	EmptyEvents				: ST_Event; // to Clear the event array[n]
	CmdEmpty				: ST_Command;
	iEventNameFailed 		: E_EventName;
	iEventName				: E_EventName;

	//nCommandNumber:UINT;
	//fbModuleIDNameCheck: FB_ModuleIDNameCheck;
	//fbParameterCheck: FB_ParameterCheck;	
END_VAR

VAR_IN_OUT
	arrRCMD 				: ARRAY [1..NO_OF_CMD_BUFFER] OF ST_Command;
	arrEvent				: ARRAY [1..NO_OF_EVENT_BUFFER] OF ST_Event;
END_VAR
//nCommandNumber := INT_TO_UINT(n);
bErr    														:= FALSE;
sStatus 														:= '';

arrEvent[n] 													:= EmptyEvents;

IF arrRCMD[n].eTaskName = E_TaskName.AlarmReset THEN
	M_nModuleIDConversion(eModuleID:=arrRCMD[n].eModuleID,iLevel=>iLevel);
	//iLevel := arrRCMD[n].iParam[1];
	//iLevel := arrRCMD[n].iParam[1]/1000;
ELSE
	M_nModuleIDConversion(eModuleID:=arrRCMD[n].eModuleID,iLevel=>iLevel);
	(*
	CASE arrRCMD[n].eModuleID OF
		E_ModuleID.TESTER_L_A_01 : iLevel:=1;
		E_ModuleID.TESTER_L_A_02 : iLevel:=2;
		E_ModuleID.TESTER_L_A_03 : iLevel:=3;
		
	END_CASE
	*)	
END_IF

IF bInvalidCommand = TRUE THEN
	bErr := TRUE; 
	sStatus := 'Invalid command received';
ELSIF iLevel = 0 THEN
	bErr := TRUE; 
	sStatus := 'Wrong Module ID';
ELSIF  arrTCShuttlePOC[iLevel].stGblParam.bAlarmOccur =TRUE THEN
	IF arrRCMD[n].eTaskName = E_TaskName.TIUSlideOut THEN 
		bErr := TRUE; 
		sStatus := 'Please clear alarm 1st';
	//ELSIF UDINT_TO_INT(arrTCVIO[iLevel].iAlarmCode) <> arrRCMD[n].iParam[1] THEN
	//	bErr := TRUE; 
	//	sStatus := concat('Alarm Code not match with current AlarmCode ', UDINT_TO_STRING(arrTCVIO[iLevel].iAlarmCode));
	END_IF
ELSIF arrRCMD[n].eTaskName = E_TaskName.TCCSessionRequest OR
   		arrRCMD[n].eTaskName = E_TaskName.DPSPower OR
   		arrRCMD[n].eTaskName = E_TaskName.TIUSlideOut THEN
			//bErr:=SEL(arrTCLevelState[iLevel] = E_State.eDisabled,FALSE,TRUE);
			//sStatus := SEL(bErr,'','Module is Disabled');
			bErr:=SEL(TC_ModuleState[iLevel].Tester = E_State.eDisabled OR 
					  TC_ModuleState[iLevel].TCSite[1].TCU = E_State.eDisabled OR 
					  TC_ModuleState[iLevel].TCSite[1].TIERII = E_State.eDisabled 
					  ,FALSE,TRUE);
			IF TC_ModuleState[iLevel].Tester = E_State.eDisabled THEN
				sStatus := SEL(bErr,'','Tester Cell Module is Disabled');
			ELSIF TC_ModuleState[iLevel].TCSite[1].TCU = E_State.eDisabled THEN
				sStatus := SEL(bErr,'','Tester Cell TCU is Disabled');
			ELSIF TC_ModuleState[iLevel].TCSite[1].TIERII = E_State.eDisabled THEN
				sStatus := SEL(bErr,'','Tester Cell TierII is Disabled');
			END_IF
END_IF

IF bErr THEN
	iSendEvent :=2;
	JMP iSendEvent;
ELSE
	arrTCShuttlePOC[iLevel].stGblParam.stTACommand := arrRCMD[n];
	
	CASE arrRCMD[n].eTaskName OF
		E_TaskName.TCCSessionRequest	: 	
			M_TCCSessionRequest(n:=n, arrRCMD:= arrRCMD, arrEvent:= arrEvent);
			//iSendEvent :=SEL(M_TCCSessionRequest(n:=n, arrRCMD:= arrRCMD, arrEvent:= arrEvent),2,1);

	
		E_TaskName.SetLogFileVerbosity	: 	
			M_SetLogfileVerbosity(n:=n, arrRCMD:= arrRCMD, arrEvent:= arrEvent);
	
		E_TaskName.EnableModule,
		E_TaskName.DisableModule:
			M_EnableModule(n:=n,arrRCMD:=arrRCMD,arrEvent:=arrEvent);
			
		E_TaskName.DoorClose:
			M_DoorOpenClose(n:=n, bLock:=TRUE, bFrontDoor:=FALSE, arrRCMD:=arrRCMD,arrEvent:=arrEvent);
		E_TaskName.DoorOpen:
			M_DoorOpenClose(n:=n, bLock:=FALSE, bFrontDoor:=FALSE, arrRCMD:=arrRCMD,arrEvent:=arrEvent);
		
		E_TaskName.DPSPower:
				//M_DPSPower(n:=n,arrRCMD:=arrRCMD,arrEvent:=arrEvent);	
				IF arrRCMD[n].iParam[1]=0 THEN
				arrTCShuttlePOC[iLevel].stGblParam.bDSPPowerOff:= TRUE;
				ELSIF arrRCMD[n].iParam[1]=1 THEN
					arrTCShuttlePOC[iLevel].stGblParam.bDSPPowerOn := TRUE;
				ELSIF arrRCMD[n].iParam[1]=2 THEN
					arrTCShuttlePOC[iLevel].stGblParam.bDSPPowerAuto := TRUE;
				END_IF	
			
		E_TaskName.TIUSlideOut : 
			//IF arrTCMultiLevel[iLevel].stGblParam.bTCCSessionReq THEN
			//	sStatus := 'Module is In Manual TCC Request Operation Session';
			//	iSendEvent :=2;
			//	JMP iSendEvent;
			//END_IF
			IF arrTCShuttlePOC[iLevel].stGblParam.iProcessStep=E_ProcessStep.eSeqError THEN
				sStatus := 'TIUSlideOUT Process Busy! Retry Or Cancel First';
				iSendEvent :=2;
				JMP iSendEvent;
			ELSIF FALSE(*Col or LvlSeq Err Or TIIErr*) THEN
				sStatus := 'Clear the alarm';
				iSendEvent :=1;
				JMP iSendEvent;
			END_IF
			IF arrRCMD[n].bParam[1]=TRUE THEN
				arrTCShuttlePOC[iLevel].stGblParam.bShuttleMoveOut := TRUE;
			ELSE
				arrTCShuttlePOC[iLevel].stGblParam.bShuttleMoveIn := TRUE;
			END_IF
		
		E_TaskName.Initialize : 	
		IF  arrTCShuttlePOC[iLevel].stGblParam.bAlarmOccur =TRUE THEN
			bErr := TRUE; 
			sStatus := 'Please clear alarm 1st';
			iSendEvent :=2;
			JMP iSendEvent;
		ELSE
			arrTCShuttlePOC[iLevel].stGblParam.bInitialise :=TRUE;
		END_IF
			
			
		E_TaskName.TIUSlideOutRetry : 	
			IF arrTCShuttlePOC[iLevel].stGblParam.iProcessStep<>E_ProcessStep.eSeqError THEN
				sStatus := 'Nothing to Retry';
				iSendEvent :=2;
				JMP iSendEvent;
			ELSIF FALSE(*Col or LvlSeq Err Or TIIErr*) THEN
				sStatus := 'Clear the alarm';
				iSendEvent :=2;
				JMP iSendEvent;
			END_IF
			IF arrTCShuttlePOC[iLevel].stGblParam.bAlarmOccur THEN
				sStatus := 'Clear the Alarm First!';
				iSendEvent :=2;
				JMP iSendEvent;
			END_IF
			arrTCShuttlePOC[iLevel].stGblParam.bResume :=TRUE;
		
		E_TaskName.Cancel : 	
			IF arrTCShuttlePOC[iLevel].stGblParam.bShuttleMoveOut=TRUE
			OR arrTCShuttlePOC[iLevel].stGblParam.bShuttleMoveIn=TRUE 
			OR arrTCMultiLevel[iLevel].stGblParam.bDSPPowerOff 
			OR arrTCMultiLevel[iLevel].stGblParam.bDSPPowerOn 
			OR arrTCMultiLevel[iLevel].stGblParam.bDSPPowerAuto 
			THEN
				arrTCShuttlePOC[iLevel].stGblParam.bCancel :=TRUE;
				arrTCShuttlePOC[iLevel].stGblParam.bInternalCancel :=TRUE;
			ELSE
				sStatus := 'Nothing to cancel';
				iSendEvent :=1;
				JMP iSendEvent;
			END_IF
			
		E_TaskName.TIUSlideOutCancel : 	
			IF arrTCShuttlePOC[iLevel].stGblParam.bShuttleMoveOut=TRUE OR arrTCShuttlePOC[iLevel].stGblParam.bShuttleMoveIn=TRUE THEN
				arrTCShuttlePOC[iLevel].stGblParam.bTIUSlideOutCancel:=TRUE;
				//arrTCShuttlePOC[iLevel].stGblParam.bInternalCancel :=TRUE;
			ELSE
				sStatus := 'Nothing to cancel';
				iSendEvent :=1;
				JMP iSendEvent;
			END_IF
				
		E_TaskName.AlarmReset : 	
			IF M_AlarmReset(n:=n, arrRCMD:=arrRCMD, arrEvent:=arrEvent) THEN
			arrTCShuttlePOC[iLevel].stGblParam.bAlarmClear :=TRUE;
			//iSendEvent :=1;
			//JMP iSendEvent;
			END_IF
			
			//arrTCShuttlePOC[iLevel].stGblParam.bAlarmClear :=TRUE;
			//iSendEvent :=1;
			//M_AlarmReset(n:=30, arrRCMD:=arrRCMD, arrEvent:=arrEvent);
			//JMP iSendEvent;
			
			//M_AlarmReset(n:=30, arrRCMD:=arrRCMD, arrEvent:=arrEvent);
		//E_TaskName.EnableModule: ;  //Set Flag 		(Bypass Alarm)
		//E_TaskName.DisableModule: ; // Reset Flag
		//E_TaskName.DoorOpen: ; // unlock door output here;
		//E_TaskName.DoorClose: ; // Door Recovery
		//arrTCShuttlePOC[iLevel].stGblParam.bDoorClose :=TRUE;
						
	END_CASE
END_IF

//send event to TA
iSendEvent :
IF iSendEvent<>0 THEN
	M_nCmdtoEvent(eCmd2Event_TaskName:=arrRCMD[n].eTaskName , iCmd2Event_Result:=iSendEvent , eCmd2Event_EventName:=iEventName , sCmd2Event_EventName:=sLogName );
	M_AddEvent(
		sLogName:= sLogName, 
		eEventName:= iEventName, 
		eModuleID:= arrRCMD[n].eModuleID, 
		iParam:= arrRCMD[n].iParam, 
		sParam:= arrRCMD[n].sParam, 
		bParam:= arrRCMD[n].bParam, 
		dParam:= arrRCMD[n].dParam, 
		sFailReason:= sStatus);
	iSendEvent :=0;
END_IF

arrRCMD[n]:= CmdEmpty;
END_METHOD

METHOD M_ProcessMLCommand : BOOL
VAR_INPUT
	n								: INT; // Array number of which 10 commands to be processed
	bInvalidCommand					: BOOL;
	bRetry 							: BOOL;
	bCancel							: BOOL;
END_VAR

VAR
	bErr							: BOOL; // var for error flag
	bFrontDoor						: BOOL;
	
	iSendEvent						: INT;
	
	i								: UINT; // variable to loop all 6 parameters
	nCommandNumber					: UINT;
	nParameterNumber				: UINT;	
	
	iLevel 							: DINT := 0;
	
	sStatus							: STRING; // var for error message
	sLogName						: STRING(81);
	str								: STRING;
	
	EmptyEvents						: ST_Event; // to Clear the event array[n]
	CmdEmpty						: ST_Command;
	iEventNameFailed 				: E_EventName;
	iEventName						: E_EventName;
	stMLVIO							: ST_TCMultiLevel_VIO;
	stColVIO						: ST_TCColumn_VIO;
	stDbStnVIO						: ST_DebugStation_VIO;
	//fbModuleIDNameCheck: FB_ModuleIDNameCheck;
	//fbParameterCheck: FB_ParameterCheck;	
END_VAR

VAR_IN_OUT
	arrRCMD 						: ARRAY [1..NO_OF_CMD_BUFFER] OF ST_Command;
	arrEvent						: ARRAY [1..NO_OF_EVENT_BUFFER] OF ST_Event;
END_VAR
/////////////////////////////////////////////////////////////////////////////////////////////////////////////////////////////////////////////////////////////////////////////////////////////////
//	
/////////////////////////////////////////////////////////////////////////////////////////////////////////////////////////////////////////////////////////////////////////////////////////////////
bErr    																		:= FALSE;
sStatus																			:= '';
bFrontDoor																		:= FALSE;
                                                            					
arrEvent[n]																		:= EmptyEvents;
                                                            					
IF arrRCMD[n].eTaskName = E_TaskName.AlarmReset THEN        					
	M_nModuleIDConversion(                                  					
		eModuleID																:= arrRCMD[n].eModuleID,
		iLevel																	=> iLevel);
ELSE                                                        						
	M_nModuleIDConversion(                                  	
		eModuleID																:= arrRCMD[n].eModuleID,
		iLevel																	=> iLevel);
	IF ilevel > 100 AND bDebugCart THEN                     					
		bFrontDoor																:= TRUE;
		iLevel																	:= iLevel - 100;
	END_IF
END_IF

IF (bDebugCart AND iLevel > 2 AND iLevel <> 99 AND NOT 100 < iLevel AND NOT iLevel < 103) THEN
	bErr																		:= TRUE;
	str																			:= '';
  	str 																		:= CONCAT(str,': Cell Level');
	str																			:= CONCAT(str,'[');
	str																			:= CONCAT(str,DINT_TO_STRING(iLevel));
	str																			:= CONCAT(str,'] ');
	sStatus																		:= 'Invalid Module ID';
	sStatus																		:= CONCAT(sStatus,str);
END_IF

IF NOT (bDebugStation OR bDebugCart) AND NOT IsNetIDReadOK THEN
	bErr																		:= TRUE;
	str																			:= '';
	sStatus																		:= 'Invalid Colum AMS Net ID, Please Set up Column AMS Net ID First ';
	sStatus																		:= CONCAT(sStatus,str);
END_IF

stMLVIO																			:= arrTCMultiLevel[iLevel].fbTCMultiLevelSeq.P_stTCMultiLevelVIO;

// Invalid command
IF bInvalidCommand = TRUE THEN
	bErr																		:= TRUE; 
	sStatus																		:= 'Invalid command received';
	
// Only cancel command allow iLevel is 0
ELSIF iLevel = 0 AND arrRCMD[n].eTaskName <> E_TaskName.Cancel THEN
	bErr																		:= TRUE; 
	sStatus																		:= 'Wrong Module ID';
	
// IO Diagnostic Mode
ELSIF bDiagnosticMode THEN
	bErr																		:= TRUE; 
	sStatus																		:= 'IO Diagnostic Mode is Enabled';
	
// Task name is TCCSessionRequest or DPSPower or TIUSlideOut
ELSIF arrRCMD[n].eTaskName = E_TaskName.TCCSessionRequest OR arrRCMD[n].eTaskName = E_TaskName.DPSPower THEN
	
	bErr																:=  TC_ModuleState[iLevel].TCSite[1].TCU = E_State.eDisabled 	OR 
			  																TC_ModuleState[iLevel].TCSite[1].TIERII = E_State.eDisabled	OR
																			TC_ModuleState[iLevel].Tester = E_State.eDisabled;
	
	IF TC_ModuleState[iLevel].Tester = E_State.eDisabled THEN
		sStatus 															:= SEL(bErr, '', 'Tester Cell Module is Disabled');
	ELSIF TC_ModuleState[iLevel].TCSite[1].TCU = E_State.eDisabled THEN
		sStatus																:= SEL(bErr, '', 'Tester Cell TCU is Disabled'); 
	ELSIF TC_ModuleState[iLevel].TCSite[1].TIERII = E_State.eDisabled THEN
		sStatus 															:= SEL(bErr, '', 'Tester Cell TierII is Disabled');
	END_IF

ELSIF arrRCMD[n].eTaskName = E_TaskName.TIUSlideOut THEN
	bErr																:= TC_ModuleState[iLevel].TCSite[1].TCU = E_State.eDisabled;
	
	IF TC_ModuleState[iLevel].Tester = E_State.eDisabled THEN
		sStatus 															:= SEL(bErr, '', 'Tester Cell Module is Disabled');
	END_IF
END_IF

//TII Alarm And System Alarm Check
// 1. Task name is not cancel
// 2. Task name is not alarm reset
// 3. Task name is not door open
// 4. Task name is not door close
// 5. Task name is not SetBlinkRate
// 6. Either no leak and ground alarm or Task name is not TIUSlideOut and DrawerUp or both
IF 	arrRCMD[n].eTaskName <> E_TaskName.Cancel 														AND 
	arrRCMD[n].eTaskName <> E_TaskName.AlarmReset 													AND 
  	arrRCMD[n].eTaskName <> E_TaskName.DoorOpen 													AND  //front OR back door open shouldnt block by any alarm
	arrRCMD[n].eTaskName <> E_TaskName.DoorClose													AND //front OR back door close shouldnt block by any alarm
	arrRCMD[n].eTaskName <> E_TaskName.SetBlinkRate 												AND
	(stMLVIO.bAlarmBlock OR stMLVIO.iSysUnBlockAlm = 2 OR stMLVIO.iSysUnBlockAlm = 10)  			THEN
	
		FOR i:= 1 TO NO_OF_COMMON_SENSOR DO
			IF ALMTC.Common.AlarmID[i] THEN
				IF sStatus = '' THEN 
					sStatus														:= SysAlmText[i];	
					CONTINUE;				
				END_IF
				sStatus															:= CONCAT(CONCAT(sStatus,', '),SysAlmText[i]);
			END_IF
		END_FOR
		
		FOR i:= 1 TO NO_OF_TII_SENSOR DO
			IF ALMTC.Level[iLevel].AlarmID[i] THEN
				IF sStatus = '' THEN 
					sStatus														:= TIIAlmText[i];	
					CONTINUE;				
				END_IF
				sStatus															:= CONCAT(CONCAT(sStatus,', '),TIIAlmText[i]);
			END_IF
		END_FOR
		
		bErr 																	:= TRUE;
END_IF

IF arrRCMD[n].eTaskName <> E_TaskName.Cancel THEN 
	IF arrTCMultiLevel[iLevel].stGblParam.bAlarmOccur = TRUE THEN
		
		IF 	arrRCMD[n].eTaskName = E_TaskName.TIUSlideOut 	OR arrRCMD[n].eTaskName = E_TaskName.DrawerUp 	OR	arrRCMD[n].eTaskName = E_TaskName.DPSPower 	OR
			arrRCMD[n].eTaskName = E_TaskName.AP240ACPOWER 	OR arrRCMD[n].eTaskName = E_TaskName.TIUSlideOutRetry THEN  
				bErr 																:= TRUE; 
				sStatus 															:= 'Please clear alarm 1st';
		END_IF
		
	ELSIF 	arrTCMultiLevel[iLevel].stGblParam.iProcessState = E_ProcessState.ePAUSE AND 
			(NOT (arrRCMD[n].eTaskName<>E_TaskName.TIUSlideOutRetry OR arrRCMD[n].eTaskName<>E_TaskName.AlarmReset)) THEN
				bErr 																:= TRUE;
				sStatus 															:= 'Clear Or Cancel The Command First';
	END_IF
END_IF	

	
IF bErr THEN
	iSendEvent 																	:= 2;
	JMP iSendEvent;
ELSE
	// Cancel Command pass in without Module ID
	IF (arrRCMD[n].eTaskName <> E_TaskName.Cancel) THEN	
		IF bDebugStation THEN
			stDebugStation.stGblDBStnParam.stTACommand 							:= arrRCMD[n];
		ELSE
			arrTCMultiLevel[iLevel].stGblParam.stTACommand 						:= arrRCMD[n]; 
		END_IF
	 END_IF
	
	CASE arrRCMD[n].eTaskName OF
		E_TaskName.SetBlinkRate: 
			M_SetBlinkRate(
				arrRCMD															:= arrRCMD, 
				arrEvent														:= arrEvent);
	
		E_TaskName.AP240ACPOWER:
			IF (NOT bDebugCart) AND arrRCMD[n].iParam[1] <> 0 AND arrTCMultiLevel[iLevel].stGblParam.bTCCellACPwrOff THEN
				sStatus 														:= 'TBotEAP_TCCCellACPowerOFF_Signal_Detected';
				bErr															:= TRUE;
				iSendEvent 														:= 2;
				JMP iSendEvent;
			END_IF
			
			IF bDebugCart AND arrRCMD[n].iParam[1] <> 0 AND DS_Facility_eapShutOffAllACPower THEN
				sStatus 														:= 'DS Facility Cell 240 AC Power OFF Signal Detected';
				bErr															:= TRUE;
				iSendEvent 														:= 2;
				JMP iSendEvent;
			END_IF
			
			IF bDebugStation AND iLevel = 1 THEN 
				IF arrRCMD[n].iParam[1] = 0 THEN
					stDebugStation.stGblDBStnParam.bAP240ACPowerOff				:= TRUE;
				ELSIF arrRCMD[n].iParam[1] = 1 THEN
					stDbStnVIO 													:= stDebugStation.fbDBStnSeq.P_stVIO;//.P_stTCMultiLevelVIO;
					IF stDbStnVIO.ipDBStnAPPresentSensor THEN
						stDebugStation.stGblDBStnParam.bAP240ACPowerOn 			:= TRUE;
					ELSE
						bErr													:= TRUE;
						IF (NOT stDbStnVIO.ipDBStnAPPresentSensor) THEN 
							sStatus 											:= 'AP is not present';
						END_IF
						iSendEvent 												:= 2;
						JMP iSendEvent;
					END_IF
				END_IF
				
			ELSE // if Not Debug station 
				IF arrRCMD[n].iParam[1] = 0 THEN
					arrTCMultiLevel[iLevel].stGblParam.bAP240ACPowerOff			:= TRUE;
				ELSIF arrRCMD[n].iParam[1] = 1 THEN
					stMLVIO 													:= arrTCMultiLevel[iLevel].fbTCMultiLevelSeq.P_stTCMultiLevelVIO;
					IF stMLVIO.ipTesterPresent AND NOT stMLVIO.ipTesterPowerOn THEN
						bErr													:= TRUE;
						sStatus													:= 'Tester power is not ON';
						iSendEvent 												:= 2;
						JMP iSendEvent;
					ELSIF (NOT stMLVIO.ipAPPresentSensor) THEN
						bErr													:= TRUE;
						sStatus													:= 'AP is not present';
						iSendEvent 												:= 2;
						JMP iSendEvent;
					ELSE
						arrTCMultiLevel[iLevel].stGblParam.bAP240ACPowerOn 		:= TRUE;
					END_IF
				END_IF
			END_IF
		
		E_TaskName.DrawerUp: 
			stMLVIO																:= arrTCMultiLevel[iLevel].fbTCMultiLevelSeq.P_stTCMultiLevelVIO;
			
			IF stMLVIO.bTCCSessionActiveStatusFlag THEN
				bErr															:= TRUE;
				sStatus															:= 'Module is In Manual TCC Request Operation Session';
				iSendEvent														:= 2;
				JMP iSendEvent;
			END_IF
			
			IF stMLVIO.ipAPPresentSensor AND (NOT stMLVIO.ipAPReady) THEN
				bErr															:= TRUE;
				sStatus															:= 'AP Ready Signal is not Detected';
				iSendEvent														:= 2;
				JMP iSendEvent;
			END_IF
			
			IF arrRCMD[n].bParam[1] = TRUE THEN
				IF ((stMLVIO.ipTCCellTbotSideDoorOpenCloseStatus01 AND stMLVIO.ipTCCellTbotSideDoorOpenCloseStatus02 AND stMLVIO.ipTCCellDoorOpenCloseStatus) OR (NOT bDebugCart)) AND 
					((stMLVIO.ipTCCellDoorOpenCloseStatus) OR bDebugCart)THEN
					arrTCMultiLevel[iLevel].stGblParam.bDrawerUp				:= TRUE;
				ELSE
					bErr														:= TRUE;
					sStatus														:= 'Please Close and Lock the Door(s) First';
					iSendEvent													:= 2;
					JMP iSendEvent;
				END_IF
			ELSE
				arrTCMultiLevel[iLevel].stGblParam.bDrawerDown					:= TRUE;
			END_IF
			
		E_TaskName.EnableModule, E_TaskName.DisableModule:	
			;
		E_TaskName.SetLogFileVerbosity:	
			;	
		E_TaskName.TCCSessionRequest: 	
			stMLVIO																:= arrTCMultiLevel[iLevel].fbTCMultiLevelSeq.P_stTCMultiLevelVIO;
			IF (NOT stMLVIO.ipTCDrawerCylRetractRS) THEN
				bErr															:= TRUE;
				sStatus															:= 'Tester Drawer is not in Retracted Position';
				iSendEvent														:= 2;
				JMP iSendEvent;
			END_IF
			
			IF (NOT stMLVIO.ipTCDrawerCylDownRS) THEN
				bErr															:= TRUE;
				sStatus															:= 'Tester Drawer is not in Down Position';
				iSendEvent														:= 2;
				JMP iSendEvent;
			END_IF
			
			M_TCCSessionRequest(
				n																:= n, 
				arrRCMD															:= arrRCMD, 
				arrEvent														:= arrEvent);
		
		E_TaskName.DoorClose:
			M_DoorOpenClose(
				n																:= n, 
				bLock															:= TRUE, 
				bFrontDoor														:= bFrontDoor, 
				arrRCMD															:= arrRCMD,
				arrEvent														:= arrEvent);
			
		E_TaskName.DoorOpen:
			M_DoorOpenClose(
				n																:= n, 
				bLock															:= FALSE,
				bFrontDoor														:= bFrontDoor, 
				arrRCMD															:= arrRCMD,
				arrEvent														:= arrEvent);					
							
		E_TaskName.TesterAirValve:
			M_AirOnOFF(
				n																:= n,
				iValSelection													:= E_AirValve.TESTER,
				arrRCMD															:= arrRCMD,
				arrEvent														:= arrEvent);
			
		E_TaskName.APAirValve:
			M_AirOnOFF(
				n																:= n,
				iValSelection													:= E_AirValve.AP,
				arrRCMD															:= arrRCMD,
				arrEvent														:= arrEvent);
			
		E_TaskName.TIUSocketCoolingAir:
			IF arrRCMD[n].iParam[1] = 1 THEN	
				M_AirOnOFF(
					n															:= n, 
					iValSelection												:= E_AirValve.TIU_SKT1, 
					arrRCMD														:= arrRCMD, 
					arrEvent													:= arrEvent);
			ELSIF arrRCMD[n].iParam[1] = 2 THEN
				M_AirOnOFF(
					n															:= n, 
					iValSelection												:= E_AirValve.TIU_SKT2, 
					arrRCMD														:= arrRCMD, 
					arrEvent													:= arrEvent);	
			ELSE
				bErr															:= TRUE;
				sStatus															:= 'Invalid TIUSocketCoolingAirParameter';
				iSendEvent														:= 2;
				JMP iSendEvent;
			END_IF
			
		E_TaskName.DPSPower:
			IF (NOT bDebugCart) AND arrRCMD[n].iParam[1] <> 0 AND arrTCMultiLevel[iLevel].stGblParam.bTCCellACPwrOff THEN
				sStatus															:= 'TBotEAP_TCCCellACPowerOFF_Signal_Detected';
				bErr															:= TRUE;
				iSendEvent														:= 2;
				JMP iSendEvent;
			END_IF
			
			IF bDebugCart AND arrRCMD[n].iParam[1] <> 0 AND DS_Facility_eapShutOffAllACPower THEN
				sStatus 														:= 'DS Facility Cell 240 AC Power OFF Signal Detected';
				bErr															:= TRUE;
				iSendEvent 														:= 2;
				JMP iSendEvent;
			END_IF
			
			// 0:OFF,1:ON,2:AUTO, ***-1:SELFLOOP,99:ALARMOCCURED
			IF arrRCMD[n].iParam[1] = 0 THEN // OFF Param
				arrTCMultiLevel[iLevel].stGblParam.bDSPPowerOff					:= TRUE;
				arrTCMultiLevel[iLevel].stGblParam.iTstPwrCmd					:= 0;
			ELSIF arrRCMD[n].iParam[1] = 1 THEN	// ON Param
				stMLVIO 														:= arrTCMultiLevel[iLevel].fbTCMultiLevelSeq.P_stTCMultiLevelVIO;
				IF stMLVIO.ipTesterPresent AND stMLVIO.ipTesterLatchesClosed THEN
					arrTCMultiLevel[iLevel].stGblParam.bDSPPowerOn 				:= TRUE;
					arrTCMultiLevel[iLevel].stGblParam.iTstPwrCmd				:= 1;
				ELSE
					bErr														:= TRUE;
					IF (NOT stMLVIO.ipTesterPresent) THEN 
						sStatus													:= 'Tester is not present';
					ELSIF (NOT stMLVIO.ipTesterLatchesClosed) THEN
						sStatus													:= 'Tester Latch is not Closed';
					END_IF
					iSendEvent													:= 2;
					JMP iSendEvent;
				END_IF
			ELSIF arrRCMD[n].iParam[1] = 2 THEN	//AUTO Param
				arrTCMultiLevel[iLevel].stGblParam.bDSPPowerAuto				:= TRUE;
			END_IF

		E_TaskName.TIUSlideOut:				
			IF arrRCMD[n].bParam[1] = TRUE THEN
				IF bDebugCart THEN
					sStatus 													:= 'Cell Not Allow to move out in Debug Cart Mode';
					iSendEvent 													:= 2;
					JMP iSendEvent;
				END_IF
				
				stColVIO														:= fbTCColumn.P_stTCColumnVIO;
				IF (NOT stColVIO.ipTbotDoorClosedSignal) AND (NOT bDebugCart) AND (NOT bDebugStation) THEN
					bErr														:= TRUE;
					sStatus														:= 'Tbot Door Not Closed.';
					ALMTC.Common.AlarmID[E_ColAlarm.ipTbotDoorClosedSignal]		:= TRUE;
					iSendEvent													:= 2;
					JMP iSendEvent;
				END_IF
				
				IF (NOT arrTCMultiLevel[iLevel].stGblParam.bTCDwrSafeToMoveEAP) THEN
					bErr														:= TRUE;
					sStatus														:= 'TBOT EAP Not allow Drawer Safe To Move.';
					iSendEvent													:= 2;
					JMP iSendEvent;
				END_IF
				
				arrTCMultiLevel[iLevel].stGblParam.bShuttleMoveOut				:= TRUE ;
			ELSE
				arrTCMultiLevel[iLevel].stGblParam.bShuttleMoveIn				:= TRUE;
			END_IF

		E_TaskName.Initialize: 	
			stColVIO														:= fbTCColumn.P_stTCColumnVIO;
			IF (NOT stColVIO.ipTbotDoorClosedSignal) AND (NOT bDebugCart) AND (NOT bDebugStation) THEN
				bErr														:= TRUE;
				sStatus														:= 'Tbot Door Not Closed.';
				ALMTC.Common.AlarmID[E_ColAlarm.ipTbotDoorClosedSignal]		:= TRUE;
				iSendEvent													:= 2;
				JMP iSendEvent;
			END_IF
			
			IF bDebugStation AND iLevel = 1 THEN 
				stDebugStation.stGblDBStnParam.bInitialise						:= TRUE;
			ELSE
				arrTCMultiLevel[iLevel].stGblParam.bInitialise					:= TRUE;
			END_IF
					
		E_TaskName.TIUSlideOutRetry: 	
			IF arrTCShuttlePOC[iLevel].stGblParam.bAlarmOccur THEN
				sStatus 														:= 'Clear the Alarm First!';
				iSendEvent 														:= 2;
				JMP iSendEvent;
			ELSE
			
			stColVIO														:= fbTCColumn.P_stTCColumnVIO;
			IF (NOT stColVIO.ipTbotDoorClosedSignal) AND (NOT bDebugCart) AND (NOT bDebugStation) THEN
				bErr														:= TRUE;
				sStatus														:= 'Tbot Door Not Closed.';
				ALMTC.Common.AlarmID[E_ColAlarm.ipTbotDoorClosedSignal]		:= TRUE;
				iSendEvent													:= 2;
				JMP iSendEvent;
			END_IF
			
			IF (NOT arrTCMultiLevel[iLevel].stGblParam.bTCDwrSafeToMoveEAP) THEN
				bErr														:= TRUE;
				sStatus														:= 'TBOT EAP Not allow Drawer Safe To Move.';
				iSendEvent													:= 2;
				JMP iSendEvent;
			END_IF

			IF arrRCMD[n].bParam[1] = TRUE THEN
				arrTCMultiLevel[iLevel].stGblParam.bShuttleMoveOut			:= TRUE ;
			ELSE
				arrTCMultiLevel[iLevel].stGblParam.bShuttleMoveIn			:= TRUE;
			END_IF
			arrTCMultiLevel[iLevel].stGblParam.bResume						:= TRUE;
			END_IF
			
		E_TaskName.TIUSlideOutCancel: 
			stColVIO														:= fbTCColumn.P_stTCColumnVIO;	
			IF (NOT stColVIO.ipTbotDoorClosedSignal) AND (NOT bDebugCart) AND (NOT bDebugStation) THEN
				bErr														:= TRUE;
				sStatus														:= 'Tbot Door Not Closed.';
				ALMTC.Common.AlarmID[E_ColAlarm.ipTbotDoorClosedSignal]		:= TRUE;
				iSendEvent													:= 2;
				JMP iSendEvent;
			END_IF
		
			IF (NOT arrTCMultiLevel[iLevel].stGblParam.bTCDwrSafeToMoveEAP) THEN
				bErr														:= TRUE;
				sStatus														:= 'TBOT EAP Not allow Drawer Safe To Move.';
				iSendEvent													:= 2;
				JMP iSendEvent;
			END_IF
			
			IF arrTCMultiLevel[iLevel].stGblParam.bShuttleMoveOut = TRUE OR arrTCMultiLevel[iLevel].stGblParam.bShuttleMoveIn = TRUE THEN
				arrTCMultiLevel[iLevel].stGblParam.bCancel 						:= TRUE;
				
			ELSE
				sStatus															:= 'Nothing to cancel';
				
			END_IF
			iSendEvent															:= 1;
			JMP iSendEvent;
				
		E_TaskName.Cancel:
			FOR i := 1 TO NO_OF_CMD_BUFFER DO
				arrTACommands.arrTACommands[i]									:=	CmdEmpty;
			END_FOR 
			
			FOR i := 1 TO NO_OF_LEVEL DO
				IF arrTCMultiLevel[i].stGblParam.iProcessState = ePause OR arrTCMultiLevel[i].stGblParam.iProcessState = eALPAUSED THEN
					arrTCMultiLevel[i].stGblParam.bBufClear 					:= TRUE;
				END_IF
			END_FOR 	
			
			iSendEvent															:= 1;
			JMP iSendEvent;
			
		E_TaskName.AlarmReset: 
			IF arrTCMultiLevel[iLevel].stGblParam.iProcessState = eALPAUSED THEN	
				IF M_AlarmReset(
					n															:= n, 
					arrRCMD														:= arrRCMD, 
					arrEvent													:= arrEvent) THEN
					arrTCMultiLevel[iLevel].stGblParam.bAlarmClear 				:= TRUE;
				END_IF
			
			ELSE
				M_AlarmReset(
					n															:= n, 
					arrRCMD														:= arrRCMD, 
					arrEvent													:= arrEvent);
			END_IF
		E_TaskName.Secondary24VPower:
			IF bDebugStation THEN
				IF arrRCMD[n].bParam[1] = 0 THEN
					stDebugStation.stGblDBStnParam.bSecondary24VPowerOff 				:= TRUE;
				ELSIF arrRCMD[n].bParam[1] = 1 THEN
					stDebugStation.stGblDBStnParam.bSecondary24VPowerON 				:= TRUE;
				END_IF
				
			ELSE
				IF arrRCMD[n].bParam[1] = 0 THEN
					arrTCMultiLevel[iLevel].stGblParam.bSecondary24VPowerOff			:= TRUE;
				ELSIF arrRCMD[n].bParam[1] = 1 THEN
					arrTCMultiLevel[iLevel].stGblParam.bSecondary24VPowerOn				:= TRUE;
				END_IF
			END_IF
//////////////////////////////////////////////////////////////////////////////////////////////////////////////////////////////////////////////////////////////////////////////////
//////////////////////// Debug Station Commands only ////////////////////////////////////
////////////////////////////////////////////////////////////////////////////////////////////////////////////////////////////////////////////////////////////////////////////////////
		E_TaskName.SetSolenoidValves:
			IF bDebugStation THEN
				M_SetSolenoidValves(
					solenoidNumber												:= arrRCMD[n].iParam,
					on															:= arrRCMD[n].bParam[1],
				);
				
				iSendEvent														:= 1;
				JMP iSendEvent;
			ELSE
				sStatus															:= 'This command only available in Debug Station mode';
				bErr															:= TRUE;
				JMP iSendEvent;
			END_IF
	END_CASE
END_IF

//send event to TA
iSendEvent:
	IF iSendEvent <> 0 THEN
		iSendEvent																:= SEL(bErr, 1, 2);
		M_nCmdtoEvent(
			eCmd2Event_TaskName													:= arrRCMD[n].eTaskName, 
			iCmd2Event_Result													:= iSendEvent, 
			eCmd2Event_EventName												:= iEventName, 
			sCmd2Event_EventName												:= sLogName );
		arrEvent[n].sLogName													:= sLogName;
		arrEvent[n].eEventName													:= iEventName; 
		arrEvent[n].eModuleID													:= arrRCMD[n].eModuleID; 
		arrEvent[n].iParam														:= arrRCMD[n].iParam;
		arrEvent[n].sParam														:= arrRCMD[n].sParam; 
		arrEvent[n].bParam														:= arrRCMD[n].bParam; 
		arrEvent[n].dParam														:= arrRCMD[n].dParam; 
		arrEvent[n].sFailReason													:= sStatus;
	END_IF

	arrRCMD[n]																	:= CmdEmpty;
END_METHOD

METHOD M_SetBlinkRate : BOOL
VAR_INPUT
END_VAR

VAR
	bBtnState					: BOOL;
	bErr						: BOOL; // var for error flag
	
	iTCCellSubModules			: INT;
	
	iLevel						: UINT	:= 0;
	i							: UINT; // variable to loop all 6 parameters
	iSendEvent					: UINT;
	
	iBtnID						: DINT;
	iBtnBlinkFreq				: DINT;
	
	sStatus						: STRING; // var for error message
	sLogName					: STRING(255);
	sModuleID					: STRING;
	
	emoduleID					: E_ModuleID;
	EmptyEvents					: ST_Event; // to Clear the event array[n]
	CmdEmpty					: ST_Command;
	requestedState				: E_State := E_State.eEnabled;
	iEventName					: E_EventName;
	stMultiLeveVIO				: ST_TCMultiLevel_VIO;
	stDBStnVIO					: ST_DebugStation_VIO;
END_VAR

VAR_IN_OUT
	arrRCMD 					: ARRAY [1..NO_OF_CMD_BUFFER] OF ST_Command;
	arrEvent					: ARRAY [1..NO_OF_EVENT_BUFFER] OF ST_Event;
END_VAR
(*===========================================
SOLID OFF 	::State=0, 	Frequency = Don’tCare
SOLID ON 	::State=1,	Frequency = 0
BLINKING  	::State=1, 	Frequency = BlinkFreq
===========================================*)
bErr																	:= FALSE;
sStatus																	:= '';

arrEvent[n] 															:= EmptyEvents;
bBtnState																:= arrRCMD[n].bParam[1];
iBtnID																	:= arrRCMD[n].iParam[1];
iBtnBlinkFreq															:= arrRCMD[n].iParam[2];

M_nModuleIDConversion(
	eModuleID															:= arrRCMD[n].eModuleID, 
	iLevel																=> iLevel);

//moduleid 
IF iLevel = 0 THEN
	bErr 																:= TRUE; 
	sStatus 															:= 'Wrong Module ID';
ELSE	
	stMultiLeveVIO 														:= arrTCMultiLevel[iLevel].fbTCMultiLevelSeq.P_stTCMultiLevelVIO;
	stDbStnVIO 															:= stDebugStation.fbDBStnSeq.P_stVIO;
	CASE iBtnID OF
		E_LED.MaintenanceBtn:
			stMultiLeveVIO.bMtnBtnLEDState								:= bBtnState;
    		stMultiLeveVIO.iMtnBtnLEDBlinkFreq							:= iBtnBlinkFreq;	
		E_LED.AbortFlowBtn:  
			stMultiLeveVIO.bAbtBtnLEDState								:= bBtnState;
    		stMultiLeveVIO.iAbtBtnLEDBlinkFreq							:= iBtnBlinkFreq;
		E_LED.DoorUnlockBtn:  
			stMultiLeveVIO.bDoorUnlockBtnLEDState						:= bBtnState;
    		stMultiLeveVIO.iDoorUnlockBtnLEDBlinkFreq					:= iBtnBlinkFreq;
		E_DBStnLED.PurgeButton:	
			stDbStnVIO.bDBStnPurgeBtnLEDState							:= bBtnState;
			stDbStnVIO.iDBStnPurgeBtnLEDBlinkFreq						:= iBtnBlinkFreq;
	END_CASE
	arrTCMultiLevel[iLevel].fbTCMultiLevelSeq.P_stTCMultiLevelVIO		:= stMultiLeveVIO;
	stDebugStation.fbDBStnSeq.P_stVIO									:= stDBStnVIO;
END_IF

//send event to TA
iSendEvent 																:= SEL(bErr, 1, 2);

M_nCmdtoEvent(
	eCmd2Event_TaskName													:= arrRCMD[n].eTaskName, 
	iCmd2Event_Result													:= iSendEvent, 
	eCmd2Event_EventName												:= iEventName, 
	sCmd2Event_EventName												:= sLogName
);
	
arrEvent[n].sLogName													:= sLogName;
arrEvent[n].eEventName													:= iEventName; 
arrEvent[n].eModuleID													:= arrRCMD[n].eModuleID; 
arrEvent[n].iParam														:= arrRCMD[n].iParam;
arrEvent[n].sParam														:= arrRCMD[n].sParam; 
arrEvent[n].bParam														:= arrRCMD[n].bParam; 
arrEvent[n].dParam														:= arrRCMD[n].dParam; 
arrEvent[n].sFailReason													:= sStatus;

arrRCMD[n]																:= CmdEmpty;
END_METHOD

METHOD M_SetLogfileVerbosity : BOOL
VAR_INPUT
	n: UINT;          //array number of which 30 commands to be processed
END_VAR
VAR
	EmptyEvents: ST_Event; // to Clear the event array[n]
	CmdEmpty: ST_Command;
	i: INT;            //temporary variable to loop all 6 parameters
	bErr: BOOL;         //temporary var for error flag
	sStatus:STRING;     //temporary var for error message


	iEventName: E_EventName;
	sLogName: STRING(255);
	iSendEvent: UINT;
	
	requestedState : E_State := E_State.eEnabled;
	
END_VAR
VAR_IN_OUT
	arrRCMD : ARRAY [1..NO_OF_CMD_BUFFER] OF ST_Command;
	arrEvent: ARRAY [1..NO_OF_EVENT_BUFFER] OF ST_Event;
END_VAR
bErr    := FALSE;
sStatus := '';

arrEvent[n] := EmptyEvents;


IF bErr THEN
	;
ELSE
	iLogVerbosity := DINT_TO_INT(arrRCMD[n].iParam[1]);
END_IF


//send event to TA
IF bErr THEN
	iSendEvent :=2;
ELSE
	iSendEvent :=1;
END_IF

M_nCmdtoEvent(eCmd2Event_TaskName:=arrRCMD[n].eTaskName , iCmd2Event_Result:=iSendEvent , eCmd2Event_EventName:=iEventName , sCmd2Event_EventName:=sLogName );
arrEvent[n].sLogName:= sLogName;
arrEvent[n].eEventName:= iEventName; 
arrEvent[n].eModuleID:= arrRCMD[n].eModuleID; 
arrEvent[n].iParam:= arrRCMD[n].iParam;
arrEvent[n].sParam:= arrRCMD[n].sParam; 
arrEvent[n].bParam:= arrRCMD[n].bParam; 
arrEvent[n].dParam:= arrRCMD[n].dParam; 
arrEvent[n].sFailReason:= sStatus;


arrRCMD[n]:= CmdEmpty;
END_METHOD

METHOD M_SetSolenoidValves : BOOL
VAR_INPUT
	solenoidNumber	: ARRAY [1..NO_OF_INT_PARAM] OF DINT;
	on				: BOOL;
END_VAR
VAR 
	i				: INT;
	noOfSolenoids	: INT := NO_OF_INT_PARAM;
	eSolenoid		: E_Solenoid;
	stDbStnVIO		: ST_DebugStation_VIO;
	iSendEvent		: INT;
END_VAR
stDbStnVIO 										:= stDebugStation.fbDBStnSeq.P_stVIO; //get

FOR i:= 1 TO noOfSolenoids DO
	IF solenoidNumber[i] <> 0 THEN
		CASE solenoidNumber[i] OF
			E_Solenoid.opDBStnMainPCWSupply:
				stDbStnVIO.opDBStnBypassAPAirSupplySol		:= on;
				
			E_Solenoid.opDBStnMainPCWReturn:
				stDbStnVIO.opDBStnMainPCWReturn				:= on;
				
			E_Solenoid.opDBStnPCWSupplyPurge:
				stDbStnVIO.opDBStnPCWSupplyPurge			:= on;
				
			E_Solenoid.opDBStnPCWAWN:
				stDbStnVIO.opDBStnPCWAWN					:= on;
				
			E_Solenoid.opDBStnSupplyAirPurge:
				stDbStnVIO.opDBStnSupplyAirPurge			:= on;
				
			E_Solenoid.opDBStnLeakFlowPCWValve:
				stDbStnVIO.opDBStnLeakFlowPCWValve			:= on;
				
			E_Solenoid.opDBStnLowFlowPCWValve:
				stDbStnVIO.opDBStnLowFlowPCWValve			:= on;
		END_CASE
	END_IF
END_FOR

 stDebugStation.fbDBStnSeq.P_stVIO			:= stDbStnVIO;	//set
END_METHOD

METHOD PUBLIC M_TACmdUpdate : BOOL
VAR_INPUT
END_VAR
VAR
	sFormatSource					: STRING;
	iLevel							: INT;
END_VAR
/////////////////////////////////////////////////////////////////////////////////////////////////////////////////////////////////////////////////////////////////////////////////////////////////
//	State machine
/////////////////////////////////////////////////////////////////////////////////////////////////////////////////////////////////////////////////////////////////////////////////////////////////

CASE iCmdStep OF 
	0: (*Idle*)
	
		(*Action*)
		
		(*Transition*)
		IF (NOT bRCMDStart) THEN
			iCmdStep 													:= 10; // receive TA command
		ELSE 
			iCmdStep 													:= 20; // rocess TA command
		END_IF
		
	10: (*receive TA command*)	
	
		(*Action*)
		bLocalRCMDarrEmpty												:= TRUE;
	
		//Check here internal local array is empty , if not wait for same
		FOR n := 1 TO .NO_OF_CMD_BUFFER DO 
			IF arrLocalRCMD[n].eTaskName <> E_TaskName.EmptyTask THEN
				bLocalRCMDarrEmpty										:= FALSE;
				EXIT;
			END_IF	
		END_FOR
		
		IF bLocalRCMDarrEmpty THEN
			// Local array empty copy from TA array and clear TA array
			FOR n := 1 TO .NO_OF_CMD_BUFFER DO
				IF arrTA_RCMD[n].eTaskName <> E_TaskName.EmptyTask THEN
					arrLocalRCMD[n]										:= arrTA_RCMD[n]; // Copy from TA -> Local
					arrTA_RCMD[n]										:= CmdEmpty ; // Clear TA array [n]
				END_IF
			END_FOR
			
			bRCMDStart													:= TRUE; // TA cmd cleared trigger ready signal
			
			//-	IntAlignmentWithTBotPNB 1/Nov/18				
			IF iTCSReady >= 1000 THEN
				iTCSReady 												:= 0;
			ELSE
				iTCSReady 												:= iTCSReady + 1;
			END_IF
			//----------------------
		END_IF
		
		bLocalRCMDarrEmpty												:= FALSE;
		
		(*Transition*)
		iCmdStep 														:= 20; // process TA command
		
	20: (*process TA command*)	
	
		(*Action*)
		FOR n := 1 TO .NO_OF_CMD_BUFFER DO
			IF arrLocalRCMD[n].eTaskName = E_TaskName.EmptyTask THEN
				; //do nothing
			ELSE 
				fbFormat(sFormat:= 'Cmd from TA[%d]', arg1:= F_UINT(n),  sOut=> sFormatSource);
				Logging.fbDebugLog.M_nLogger(iLogLevel:= Logging.fbDebugLog.P_iLogVerbosity, sSource:= sFormatSource, sMessage:= arrLocalRCMD[n].sLogName);
				
				CASE arrLocalRCMD[n].eTaskName OF		
					E_TaskName.ActivateRecipe:	
						M_ActivateRecipe(
							n											:= n, 
							arrRCMD										:= arrLocalRCMD, 
							arrEvent									:= arrLocalEvent
						);
						
					E_TaskName.ValidateRecipe:	
						M_ValidateRecipe(
							n											:= n, 
							arrRCMD										:= arrLocalRCMD, 
							arrEvent									:= arrLocalEvent
						);
						
					E_TaskName.SetLogFileVerbosity:	
						M_SetLogfileVerbosity(
							n											:= n, 
							arrRCMD										:= arrLocalRCMD, 
							arrEvent									:= arrLocalEvent
						);
			
					E_TaskName.EnableModule, E_TaskName.DisableModule:	
						M_EnableModule(
							n											:= n,
							arrRCMD										:= arrLocalRCMD,
							arrEvent									:= arrLocalEvent
						);
					
					E_TaskName.SetBlinkRate, 		E_TaskName.TCCSessionRequest, 	E_TaskName.AlarmReset, 	E_TaskName.Resume, 			E_TaskName.Cancel,		
					E_TaskName.TIUSlideOutRetry,	E_TaskName.TIUSlideOutCancel, 	E_TaskName.Initialize, 	E_TaskName.DPSPower, 		E_TaskName.TIUSlideOut, 
					E_TaskName.DoorClose, 			E_TaskName.DoorOpen,			E_TaskName.APAirValve, 	E_TaskName.TesterAirValve, 	E_TaskName.TIUSocketCoolingAir,		
					E_TaskName.AP240ACPOWER,		E_TaskName.DrawerUp,			E_TaskName.Secondary24VPower,						E_TaskName.SetSolenoidValves:
					
						M_ProcessMLCommand(
							n											:= n, 
							arrRCMD										:= arrLocalRCMD,
							arrEvent									:= arrLocalEvent,
							bInvalidCommand								:= FALSE,
							bRetry										:= FALSE,
							bCancel										:= FALSE
						);
					
				ELSE 
					M_ProcessMLCommand(
						n												:= n, 
						arrRCMD											:= arrLocalRCMD,
						arrEvent										:= arrLocalEvent,
						bInvalidCommand									:= TRUE,
						bRetry											:= FALSE,
						bCancel											:= FALSE
					);
				END_CASE
				
				arrLocalRCMD[n]											:= CmdEmpty;
			END_IF
		END_FOR
		
		iAction															:= 1;	
		
		(*Transition*)
		iCmdStep														:= 0;		
END_CASE
END_METHOD

METHOD M_TAEventUpdate : BOOL
VAR_INPUT
END_VAR


VAR
	sFormatOut: STRING(255);
	sFormatSource : STRING(255);
	sLogName: STRING(255);
	sModuleID: STRING(255);
	sParameterStr: STRING;
END_VAR


CASE iEvtStep OF 
0: 	IF NOT bEventsStart THEN
		iEvtStep :=10; //process TA event
   	ELSE 
		iEvtStep :=20;
	END_IF
	
10: //process TA event	
	bLocalEventArrEmpty:= TRUE;
	bLocalPendingEventArrEmpty:= TRUE;

	//Collect local events (and clear previous TA events as well) 
	FOR n := 1 TO NO_OF_EVENT_BUFFER DO
	IF  arrLocalEvent[n].eEventName <> E_EventName.EmptyEvent THEN
			sModuleID := M_nModuleIDConversion(eModuleID:=arrLocalEvent[n].eModuleID);
			(*
			//sParameterStr := F_TAParamtoStr(iParam, sParam, bParam);
			fbFormat(sFormat:= '%s[%d],%s[%d]', arg1:= F_String(arrLocalEvent[n].sLogName), arg2:= F_Int(arrLocalEvent[n].eEventName), arg3:=F_String(sModuleID), 
					arg4:= F_DInt(arrLocalEvent[n].eModuleID), sOut=> sLogName ); 
			fbFormat(sFormat:= '%s,%s', arg1:= F_String(sLogName), arg2:= F_String(arrLocalEvent[n].sFailReason), sOut=> sFormatOut ); //logging
			*)
			
	sParameterStr := F_TAParamtoStr(arrLocalEvent[n].iParam, arrLocalEvent[n].sParam, arrLocalEvent[n].bParam);
	fbFormat(sFormat:= '%s[%d],%s[%d],%s', arg1:= F_String(arrLocalEvent[n].sLogName), arg2:= F_Int(arrLocalEvent[n].eEventName), arg3:=F_String(sModuleID), 
					arg4:= F_DInt(arrLocalEvent[n].eModuleID), arg5:=F_String(sParameterStr),sOut=> sLogName ); 
	fbFormat(sFormat:= '%s,%s', arg1:= F_String(sLogName), arg2:= F_String(arrLocalEvent[n].sFailReason), sOut=> sFormatOut ); //logging
			arrLocalEvent[n].sLogName:=sLogName;
			//fbFormat(sFormat:= '%s,%s', arg1:= F_String(arrLocalEvent[n].sLogName), arg2:= F_String(arrLocalEvent[n].sFailReason), sOut=> sFormatOut ); //logging
			fbFormat(sFormat:= 'Event TO TA[%d]', arg1:= F_UINT(n),  sOut=> sFormatSource);
			Logging.fbDebugLog.M_nLogger(iLogLevel:= Logging.fbDebugLog.P_iLogVerbosity, sSource:= sFormatSource, sMessage:=sFormatOut);
			arrTA_Events[n] := arrLocalEvent[n]; // Move Local[n]Event -> array TAEevnt
			arrLocalEvent[n] := EmptyEvents; // Clear Local event array[n]
			bLocalEventArrEmpty:= FALSE;
		ELSIF arrTA_Events[n].eEventName <> E_EventName.EmptyEvent THEN
			arrTA_Events[n] := EmptyEvents; // Clear previous TA Event array[n]
		END_IF
		
	END_FOR
	
	IF NOT bLocalEventArrEmpty THEN
		bEventsStart:= TRUE; //Tell TA there are events to be cleared before we will process the local pending events

//-	Int Flag 1/Nov/18
	IF iTCSEventTriggered >= 1000 THEN
		iTCSEventTriggered := 0;
	ELSE
		iTCSEventTriggered := iTCSEventTriggered + 1;
	END_IF
	//---------------------------------------------------		
		
		iEvtStep :=20;
		RETURN;
	END_IF
	
	//Check if there are local pending events
	IF arrPendingEventsQueue.Count > 0 THEN
		bLocalPendingEventArrEmpty:=FALSE;
	END_IF
	
	IF NOT bLocalPendingEventArrEmpty AND NOT bEventsUpdating THEN
	
		bEventsUpdating := TRUE; //lock it, ensure no one will read and write during updating the GVL 'arrPendingEventsQueue'
		
		iEventQueueCount   := arrPendingEventsQueue.Count;
		iEventProcessCount := arrPendingEventsQueue.Count;
	IF iEventQueueCount > NO_OF_EVENT_BUFFER THEN
		iEventProcessCount := NO_OF_EVENT_BUFFER; 
	ELSIF iEventQueueCount >= 1 THEN
		iEventProcessCount := iEventQueueCount; 	
	ELSIF iEventQueueCount < 1 THEN //In case of race condition
		//F_WriteLogWarning(WarningMessage:='Event queue buffer count is less than 1 during event processing');
		arrPendingEventsQueue.Count := 0;
		bEventsUpdating := FALSE; //release
		iEvtStep :=20;
		RETURN;
	END_IF
	
	//Collect the local pending events	
	FOR n := 1 TO iEventProcessCount DO
			arrTA_Events[n] := arrPendingEventsQueue.Queue[n]; // Copy LocalPending[n]Event -> array TAEevnt
		fbFormat(sFormat:= '%s,%s', arg1:= F_String(arrTA_Events[n].sLogName), arg2:= F_String(arrTA_Events[n].sFailReason), sOut=> sFormatOut ); //logging
		fbFormat(sFormat:= 'Event TO TA[%d]', arg1:= F_UINT(n),  sOut=> sFormatSource);
		Logging.fbDebugLog.M_nLogger(iLogLevel:= Logging.fbDebugLog.P_iLogVerbosity, sSource:= sFormatSource, sMessage:=sFormatOut);
		IF iEventQueueCount <= NO_OF_EVENT_BUFFER THEN //clear after processing (if iEventQueueCount > 10, need to dequeue)
			arrPendingEventsQueue.Queue[n] := EmptyEvents; // Clear LocalPending event array[n]
		END_IF
	END_FOR
	
	//Dequeue
	IF iEventQueueCount > NO_OF_EVENT_BUFFER THEN
		//Shift up and clear
		FOR n := NO_OF_EVENT_BUFFER+1 TO iEventQueueCount DO
			arrPendingEventsQueue.Queue[n-NO_OF_EVENT_BUFFER] := arrPendingEventsQueue.Queue[n];
			arrPendingEventsQueue.Queue[n] := EmptyEvents; 
		END_FOR
	END_IF

	arrPendingEventsQueue.Count := iEventQueueCount - iEventProcessCount;	

	bEventsUpdating := FALSE; //release
	bEventsStart:= TRUE; //Tell TA there are pending events to be cleared

//-	Int Flag 1/Nov/18
	IF iTCSEventTriggered >= 1000 THEN
		iTCSEventTriggered := 0;
	ELSE
		iTCSEventTriggered := iTCSEventTriggered + 1;
	END_IF
	//---------------------------------------------------
	
	iEvtStep :=20;
	RETURN;

END_IF

	iEvtStep :=20;
	
20: IF bEventsStart = FALSE THEN //only proceed to process the next arrLocalRCMD when the TA has cleared the bEventsStart flag to false
		iAction := 0;
	END_IF
	iEvtStep :=0;	
END_CASE
END_METHOD

METHOD M_TCCSessionRequest : BOOL
VAR_INPUT
	n: INT;        //array number of which 10 commands to be processed
END_VAR
VAR
	eProcessState:E_ProcessState	:= E_ProcessState.eUNKNOWN;
	bSessionStartEnd				: BOOL;
   	iLevel:UINT;
	EmptyEvents: ST_Event; // to Clear the event array[n]
	CmdEmpty: ST_Command;
	i: UINT;            //temporary variable to loop all 6 parameters
	bErr: BOOL;         //temporary var for error flag
	sStatus:STRING;     //temporary var for error message

	iEventName: E_EventName;
	sLogName: STRING(255);
	iSendEvent: UINT;
	stMultiLeveVIO : ST_TCMultiLevel_VIO;
	//stCommonVIO : ST_CommonSeq_VIO;
END_VAR
VAR_IN_OUT
	arrRCMD : ARRAY [1..NO_OF_CMD_BUFFER] OF ST_Command;
	arrEvent: ARRAY [1..NO_OF_EVENT_BUFFER] OF ST_Event;
END_VAR
//If NoError
	//If !OngoingProcess
		//if IsSafeForTCCRequest
			//SetTCCRequestFlagOnGlobalTA
//else 
	//Fail Request;
	
bErr    := FALSE;
sStatus := '';

arrEvent[n] := EmptyEvents;

M_nModuleIDConversion(eModuleID:=arrRCMD[n].eModuleID , iLevel=>iLevel);	
bSessionStartEnd													:= arrRCMD[n].bParam[1]; //Get Val Directly From Cmd Parameters

//moduleid 
IF iLevel =0 THEN
	bErr := TRUE; 
	sStatus := 'Wrong Module ID';
	M_TCCSessionRequest:=FALSE;
ELSE
	//eProcessState:=SEL(iPOC_ML_Selection=1,arrTCMultiLevel[iLevel].stGblParam.iProcessState,arrTCShuttlePOC[iLevel].stGblParam.iProcessState );
	eProcessState:=arrTCMultiLevel[iLevel].stGblParam.iProcessState;
	IF  eProcessState = E_ProcessState.eUNKNOWN THEN
		bErr := TRUE; 
		sStatus := ' Module is in Unknown State!';
		M_TCCSessionRequest:=FALSE;
	ELSIF  eProcessState <> E_ProcessState.eAWAITGCMD THEN
		bErr := TRUE; 
		sStatus := ' Module is Busy!';
		M_TCCSessionRequest:=FALSE;
	ELSE
		//arrTCMultiLevel[iLevel].stGblParam.bTCCSessionReq := bSessionStartEnd;  		//update to TCC Internal Global Bit
		stMultiLeveVIO:=arrTCMultiLevel[iLevel].fbTCMultiLevelSeq.P_stTCMultiLevelVIO;
		stMultiLeveVIO.bTCCSessionActiveStatusFlag := bSessionStartEnd;					//update TCCAlive Bit
		arrTCMultiLevel[iLevel].fbTCMultiLevelSeq.P_stTCMultiLevelVIO:=stMultiLeveVIO;
		M_TCCSessionRequest:=TRUE;
	END_IF
	
END_IF

//send event to TA
iSendEvent := SEL(bErr, 1, 2);
M_nCmdtoEvent(eCmd2Event_TaskName:=arrRCMD[n].eTaskName , iCmd2Event_Result:=iSendEvent , eCmd2Event_EventName:=iEventName , sCmd2Event_EventName:=sLogName );
	arrEvent[n].sLogName:= sLogName;
	arrEvent[n].eEventName:= iEventName; 
	arrEvent[n].eModuleID:= arrRCMD[n].eModuleID; 
	arrEvent[n].iParam:= arrRCMD[n].iParam;
	arrEvent[n].sParam:= arrRCMD[n].sParam; 
	arrEvent[n].bParam:= arrRCMD[n].bParam; 
	arrEvent[n].dParam:= arrRCMD[n].dParam; 
	arrEvent[n].sFailReason:= sStatus;

arrRCMD[n]:= CmdEmpty;
END_METHOD

METHOD M_ValidateRecipe : BOOL
VAR_INPUT
	n: UINT;          //array number of which 30 commands to be processed
END_VAR
VAR
	iLevel : INT := 0;
	EmptyEvents: ST_Event; // to Clear the event array[n]
	CmdEmpty: ST_Command;
	i: UINT;            //temporary variable to loop all 6 parameters
	bErr: BOOL;         //temporary var for error flag
	sStatus:STRING;     //temporary var for error message

	iEventName: E_EventName;
	sLogName: STRING(81);
	iSendEvent: UINT;
	iModuleID: DINT;
	sModuleID:STRING;
END_VAR
VAR_IN_OUT
	arrRCMD : ARRAY [1..NO_OF_CMD_BUFFER] OF ST_Command;
	arrEvent: ARRAY [1..NO_OF_EVENT_BUFFER] OF ST_Event;
END_VAR
bErr    := FALSE;
sStatus := '';

arrEvent[n] := EmptyEvents;
sModuleID := M_nModuleIDConversion(eModuleID:=arrRCMD[n].eModuleID,iLevel=>iModuleID);
sStatus:= sModuleID;
bErr:=SEL(iModuleID=0, FALSE, TRUE);

iSendEvent := SEL(bErr, 1, 2);
M_nCmdtoEvent(eCmd2Event_TaskName:=arrRCMD[n].eTaskName , iCmd2Event_Result:=iSendEvent , eCmd2Event_EventName:=iEventName , sCmd2Event_EventName:=sLogName );
arrEvent[n].sLogName:= sLogName;
arrEvent[n].eEventName:= iEventName; 
arrEvent[n].eModuleID:= arrRCMD[n].eModuleID; 
arrEvent[n].iParam:= arrRCMD[n].iParam;
arrEvent[n].sParam:= arrRCMD[n].sParam; 
arrEvent[n].bParam:= arrRCMD[n].bParam; 
arrEvent[n].dParam:= arrRCMD[n].dParam; 
arrEvent[n].sFailReason:= sStatus;
		
arrRCMD[n]:= CmdEmpty;
END_METHOD

METHOD TCUSafeState : BOOL
VAR_INPUT
	n							: INT; //array number of which 10 commands to be processed
	//bOn 						: BOOL; // true = on, false = off;
END_VAR

VAR
	sMessage					: STRING;
	sDebugSource				: STRING;
   	iLevel						: UINT;

	EmptyEvents					: ST_Event; // to Clear the event array[n]
	CmdEmpty					: ST_Command;
	i							: UINT; // variable to loop all 6 parameters
	bErr						: BOOL; // var for error flag
	sStatus						: STRING; // var for error message

	iEventName					: E_EventName;
	sLogName					: STRING(255);
	iSendEvent					: UINT;
	stMultiLeveVIO				: ST_TCMultiLevel_VIO;
	//stCommonVIO				: ST_CommonSeq_VIO;
END_VAR

VAR_IN_OUT
	arrRCMD						: ARRAY [1..NO_OF_CMD_BUFFER] OF ST_Command;
	arrEvent					: ARRAY [1..NO_OF_EVENT_BUFFER] OF ST_Event;
END_VAR
bErr											:= FALSE;
sStatus											:= '';

arrEvent[n]										:= EmptyEvents;

M_nModuleIDConversion(
	eModuleID									:= arrRCMD[n].eModuleID, 
	iLevel										=> iLevel);

//moduleid 
IF iLevel = 0 THEN
	bErr 										:= TRUE; 
	sStatus 									:= 'Wrong Module ID';
ELSE
	IF arrTCMultiLevel[iLevel].stGblParam.iProcessState = E_ProcessState.eINIT THEN
		bErr 									:= TRUE; 
		sStatus 								:= 'System initialising';
	ELSE
		fbTCUSafeState.Execute(
			n									:= n,
			iLevel								:= iLevel,
			arrRCMD								:= arrRCMD,
			arrEVENT							:= arrEVENT);;
	END_IF
END_IF

//send event to TA
iSendEvent 										:= SEL(bErr, 1, 2);

M_nCmdtoEvent(
	eCmd2Event_TaskName							:= arrRCMD[n].eTaskName, 
	iCmd2Event_Result							:= iSendEvent, 
	eCmd2Event_EventName						:= iEventName, 
	sCmd2Event_EventName						:= sLogName);
	
arrEvent[n].sLogName							:= sLogName;
arrEvent[n].eEventName							:= iEventName; 
arrEvent[n].eModuleID							:= arrRCMD[n].eModuleID; 
arrEvent[n].iParam								:= arrRCMD[n].iParam;
arrEvent[n].sParam								:= arrRCMD[n].sParam; 
arrEvent[n].bParam								:= arrRCMD[n].bParam; 
arrEvent[n].dParam								:= arrRCMD[n].dParam; 
arrEvent[n].sFailReason							:= sStatus;
arrRCMD[n]										:= CmdEmpty;
END_METHOD

END_FUNCTION_BLOCK

(* stored: Version 1.1.0.1, ProductVersion 3.1.4022.18
   POU FB_CmdAndEventUpdate: Id {595e4cc8-dfbc-4125-b9a2-14af098b52a9}, SpecialFunc None
   Method CheckTaskName: Id {d4117357-0a71-469d-8923-f3eceae84974}
   Method M_ActivateRecipe: Id {b4c781e7-fdb3-4de0-9ec0-ea2fea806a38}
   Method M_AddEvent: Id {e4098936-bc68-437a-988c-fe80ffefb0f7}
   Method M_AirOnOFF: Id {6907077e-7d9d-4836-960a-af17c54f3810}
   Method M_AlarmReset: Id {10afc52e-c32f-4a7b-9ba4-29ad15c4dab3}
   Method M_DoorOpenClose: Id {b5e53960-eb00-45b9-aef2-b703945bd1f9}
   Method M_EnableModule: Id {5ca64729-da6a-40e5-bf34-742dfdf88fdb}
   Method M_EnDisSubModuleIDConversion: Id {8206969f-b1c6-4317-a25b-10462f2b58e8}
   Method M_nCmdtoEvent: Id {67481b51-7b35-4ac2-900a-38f4d5b3ff0d}
   Method M_nModuleIDConversion: Id {16eb203b-0a4b-46dc-935c-22412fe405a9}
   Method M_ProcessCommand: Id {e97292e4-4841-4fe8-9e2e-b7f6528d13b1}
   Method M_ProcessMLCommand: Id {b788fb44-6e54-4808-b59f-702e9ec209fd}
   Method M_SetBlinkRate: Id {254ef2c7-9e83-4587-becc-f595e5487e74}
   Method M_SetLogfileVerbosity: Id {50a04445-d5e5-42f3-8cd7-3e40f6eb187f}
   Method M_SetSolenoidValves: Id {1092b1bf-9dd4-4277-b944-287bdc3d14c4}
   Method M_TACmdUpdate: Id {2a8d546c-b654-40f6-8577-b878ee586620}
   Method M_TAEventUpdate: Id {127e5a43-8677-442d-8f53-dddebd421447}
   Method M_TCCSessionRequest: Id {4d3fafa3-9931-494f-9e54-440b970cfac1}
   Method M_ValidateRecipe: Id {2994feec-8ac2-4d13-81b0-be18df259cdd}
   Method TCUSafeState: Id {98dd75fc-52a8-4c0e-9183-73eaf12b54ba} *)
